FUNCTION_BLOCK SensMsg (* Basic FB with empty ECC *)
  (* Standard: 61499-2 *)
  (* Version 1.0, 2021-03-23, dummy *)
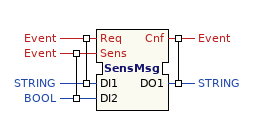
  EVENT_INPUT
    Req WITH DI1;
    Sens WITH DI2;
  END_EVENT
  EVENT_OUTPUT
    Cnf WITH DO1;
  END_EVENT
  VAR_INPUT
    DI1 : STRING;
    DI2 : BOOL;
  END_VAR
  VAR_OUTPUT
    DO1 : STRING;
  END_VAR
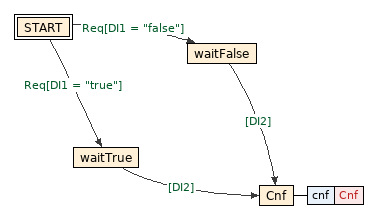
  EC_STATES
    START; (* Initial State *)
    waitTrue;
    waitFalse;
    Cnf : cnf -> Cnf;
  END_STATES
  EC_TRANSITIONS
    START TO waitTrue := Req[DI1 = "true"];
    START TO waitFalse := Req[DI1 = "false"];
    waitTrue TO Cnf := [DI2];
    waitFalse TO Cnf := [DI2];
  END_TRANSITIONS
  ALGORITHM cnf IN ST:
DO1 := DI1;
  END_ALGORITHM
END_FUNCTION_BLOCK
